(* Logix 5000 project; controller PRU vendor 1 type 14 code 107 rev 20.13; software revision 20.01 *)

TASK FeatureAdd1 (periodic, rate 10 ms, priority 10, watchdog 500 ms)
TASK INTERRUPT (periodic, rate 10 ms, priority 1, watchdog 200 ms) : SCREW_CONTROL
TASK MainTask (continuous, watchdog 500 ms) : MainProgram
TASK MSG (periodic, rate 500 ms, priority 10, watchdog 500 ms) : MSG
TASK Totalizers (periodic, rate 1000 ms, priority 3, watchdog 500 ms) : Totalizers

MODULES
   Local : vendor 1 type 14 code 107 (Compact 0, rev 20.13)
      LDI_2 : vendor 1 type 7 code 82 (Compact 15, rev 1.1, Input RPI 20 ms)
      LDI_1 : vendor 1 type 7 code 82 (Compact 14, rev 1.1, Input RPI 20 ms)
      ENCL : 1769-IQ16 (Compact 9, rev 1.1, Input RPI 2 ms)
      ENCR : 1769-IQ16 (Compact 10, rev 1.1, Input RPI 2 ms)
      LTC_3 : vendor 58 type 10 code 41 (Compact 8, rev 2.1, Input RPI 20 ms)
      LTC_4 : vendor 58 type 10 code 41 (Compact 11, rev 2.1, Input RPI 20 ms)
      LTC_2 : vendor 58 type 10 code 41 (Compact 7, rev 2.1, Input RPI 20 ms)
      LAO_1 : vendor 1 type 10 code 40 (Compact 4, rev 2.1, Output RPI 80 ms)
      LAI_1 : 1769-IF8 (Compact 1, rev 1.1, Output RPI 80 ms)
      LAI_2 : 1769-IF8 (Compact 2, rev 1.1, Output RPI 80 ms)
      LAO_2 : vendor 1 type 10 code 40 (Compact 5, rev 2.1, Output RPI 80 ms)
      LDO_2 : 1769-OB16 (Compact 13, rev 2.1, Output RPI 20 ms)
      LTC_1 : vendor 58 type 10 code 41 (Compact 6, rev 2.1, Input RPI 20 ms)
      LAI_3 : 1769-IF8 (Compact 3, rev 1.1, Output RPI 80 ms)
      LDO_1 : 1769-OB16 (Compact 12, rev 2.1, Output RPI 20 ms)
      IFS : vendor 1 type 14 code 107 (Ethernet 192.168.20.127, rev 20.1, $2b42fd4a$ RPI 500 ms)
      UTL_ENBT : 1768-ENBT (Ethernet 192.168.20.20, rev 4.1)
         UTL : vendor 1 type 14 code 74 (1768Ctrl5Slot 0, rev 20.1, $5e952958$ RPI 500 ms)
      CSS_A_ENBT : 1768-ENBT (Ethernet 192.168.20.70, rev 4.1)
         CSS_A : vendor 1 type 14 code 74 (1768Ctrl5Slot 0, rev 20.1, $71a6b3db$ RPI 500 ms)
      VFD_DRYERL : vendor 1 type 123 code 50 (Ethernet 192.168.20.112, rev 5.1, Output RPI 80 ms)
          : vendor 1 type 123 code 1535 (DPI 1, rev 6.1)
          : vendor 1 type 123 code 8192 (DPI 5, rev 4.2)
      VFD_DRYERR : vendor 1 type 123 code 50 (Ethernet 192.168.20.113, rev 5.1, Output RPI 80 ms)
          : vendor 1 type 123 code 1535 (DPI 1, rev 6.1)
          : vendor 1 type 123 code 8192 (DPI 5, rev 4.2)
      VFD_COOLSCREW : vendor 1 type 127 code 40 (Ethernet 192.168.20.114, rev 6.2, Output RPI 20 ms)
          : vendor 1 type 127 code 33792 (DSI 1, rev 1.8)
      IND560 : ETHERNET-MODULE (Ethernet 192.168.20.100, rev 1.1, Output RPI 100 ms)   // OutFeed Scale
END_MODULES

TYPE AnalogControl :
STRUCT
   AUTO : BOOL;   // 1=Auto, Control Requires automatic interlocks to enable the output
   MANUAL : BOOL;   // 1=Manual, Control (Forces the output Enable)
   MAN_SP : REAL;   // Sets the output in percent when the Manual bit is set
   AUTO_SP : REAL;   // Setpoint (usually provided by user) to control to when in Auto in Engineering Units
   CO : REAL;   // Control Output (%)
   FB : REAL;   // Feedback from the instrument (in Engineering units)
   PID_CO : REAL;   // Associated PID's Control Output (%)
   PV_SETPOINT : REAL;
   PV : REAL;   // Process Variable from measuring instrument (in Engineering units)
   HC_FAULT : BOOL;   // Controller Fault alarm bit
   RUN_STATUS : BOOL;   // Boolean feedback of the running status of the associated output
   START : BOOL;   // Master logical bit used to enable an associated output
   XA_Low : BOOL;   // Analog Signal failure (Low counts)
   XA_High : BOOL;   // Analog Signal failure (High counts)
   RawCounts : DINT;   // Raw integer from input card
   FailMode : DINT;   // In the event of a signal loss, 0=allow raw signal, 1=hold last good value, 2=hold at safe state value
   SafeState : REAL;   // Programatically set value to hold the signal to in case of a signal loss alarm
   AI_Anal : AI_Analysis;   // Used to manage an analog input to determine scaled value and loss of signal alarms
   InputMin : DINT;   // Input card lower counts i.e. 4mA - 4000 counts
   InputMax : DINT;   // Input card upper counts i.e. 20mA - 20000 counts
   ScaledMin : REAL;   // Analog low Engineering unit i.e. 4mA - 0 psi
   ScaledMax : REAL;   // Analog High Engineering unit i.e. 20mA - 100 psi
   OutputMin : DINT;   // Output card lower counts i.e. 4mA - 4000 counts
   OutputMax : DINT;   // Output card upper counts i.e. 4mA - 4000 counts
   AlarmsSetDetaults : BOOL;   // reloads the default alarm limits and setup
   Simulate : BOOL;   // 0=raw counts from Input card, 1=simulation raw counts
   RawCountsSim : DINT;   // raw count simulation from HMI/Programmer
   DifferenceExists : BOOL;   // 1 = A difference between default and current settings
   LoadDefaults : BOOL;   // set to 1=Load default values into the current values
   StoreDefaults : BOOL;   // set to 1=store the current setting values into the default settings
   AlarmDisable : BOOL;   // disables alarms 0=enabled 1=disabled
   PID_Enabled : BOOL;   // Tells the HMI if a PID exists
   mA : REAL;   // mA from Raw Counts
   AlarmWord : DINT;   // base2 alarm status
   Interlock : DINT;   // base2 Interlock Status
   HHEnabled : BOOL;
   HEnabled : BOOL;
   LEnabled : BOOL;
   LLEnabled : BOOL;
   Power : REAL;   // Current Power in kwatts
   Energy : REAL;   // Total Energy in kW-hr
   kWh_Tmr : TIMER;   // Energy Totalizer sample timer
   kWh_ResetPB : BOOL;   // HMI Reset Energy totals
   kWh_SampleTime : REAL;   // in seconds
   kWh_TimeMultiplier : REAL;   // derived from the SampleTime to ensure kW-Hr units
   PowerMax : REAL;   // Max Power Limit (kW)
END_STRUCT
END_TYPE

TYPE DateTime :   // Date and TimeOfDay (absolute) or Time (duration/interval)
STRUCT
   Yr : DINT;   // Year(s)
   Mo : DINT;   // Month(s)
   Da : DINT;   // Day(s)
   Hr : DINT;   // Hour(s)
   Min : DINT;   // Minute(s)
   Sec : DINT;   // Second(s)
   uSec : DINT;   // Microsecond(s)
END_STRUCT
END_TYPE

TYPE DUAL_SCREW :
STRUCT
   RPM_Setpoint : REAL;
   MODE_SCREW_AUTO : BOOL;
   MODE_SCREW_MAN : BOOL;
   MODE_SCREW_OFF : BOOL;
   MODE_SCREW : INT;
   SHUTDOWN_FAULTS_IOK : BOOL;
   HMI_AUTO_START_SCREW_PB : BOOL;
   HMI_STOP_SCREW_PB : BOOL;
   CMD_LEFT_SCREW_START : BOOL;
   CMD_LEFT_SCREW_STOP : BOOL;
   CMD_LEFT_SCREW_FWD : BOOL;
   CMD_LEFT_SCREW_REV : BOOL;
   CMD_RIGHT_SCREW_START : BOOL;
   CMD_RIGHT_SCREW_STOP : BOOL;
   CMD_RIGHT_SCREW_FWD : BOOL;
   CMD_RIGHT_SCREW_REV : BOOL;
   HMI_AUTO_SCREW_CMD_PCNT : REAL;
   AUTO_SCREW_LEFT_CMD_FREQ : REAL;
   AUTO_SCREW_MAX_PCNT : REAL;
   RPM_FREQ_MULTIPLIER : REAL;
   WIPER_OSC_INDEX : REAL;
   WIPER_OSC_SETPOINT : REAL;
   WIPER_OSC_AMPLITUDE : REAL;
   AUTO_SCREW_RIGHT_CMD_PCNT : REAL;
   AUTO_SCREW_RIGHT_CMD_FREQ : REAL;
   LEFT_ENCODER_G : INT;
   LEFT_ENCODER_BIN : DINT;
   RIGHT_ENCODER_G : INT;
   RIGHT_ENCODER_BIN : DINT;
   LEFT_ENCODER_TEMP : REAL;
   LEFT_ENCODER_DEG_IS : REAL;
   LEFT_ENCODER_DEG_WAS : REAL;
   RIGHT_ENCODER_TEMP : REAL;
   RIGHT_ENCODER_DEG_IS : REAL;
   RIGHT_ENCODER_DEG_WAS : REAL;
   LEFT_RIGHT_ENCODER_ERROR_TEMP : REAL;
   LEFT_RIGHT_ENCODER_ERROR_DEG : REAL;
   LEFT_ENCODER_DEG_WAS_SCANRATE : REAL;
   LEFT_ENCODER_DEG_WAS_SCANRATE_MOVED : REAL;
   RIGHT_ENCODER_DEG_WAS_SCANRATE : REAL;
   RIGHT_ENCODER_DEG_WAS_SCANRATE_MOVED : REAL;
   FINAL_SCREW_POSITION_ERROR : REAL;
   RIGHT_SCREW_RPM_COMPENSATION_GAIN : REAL;
   RIGHT_SCREW_RPM_COMP_PER_DEGREE : REAL;
   LEFT_AUTO_PCNT_SETPOINT : REAL;
   RIGHT_MAX_COMP_PCNT : REAL;
   RIGHT_MIN_COMP_PCNT : REAL;
END_STRUCT
END_TYPE

TYPE EnergyTot :   // Energy Totalizer
STRUCT
   EI : REAL;   // Current Amps
   Power : REAL;   // Current Power in kwatts
   Energy : REAL;   // Total Energy in kW-hr
   kWh_Tmr : TIMER;   // Energy Totalizer sample timer
   kWh_ResetPB : BOOL;   // HMI Reset Energy totals
   kWh_SampleTime : REAL;   // in seconds
   kWh_TimeMultiplier : REAL;   // derived from the SampleTime to ensure kW-Hr units
END_STRUCT
END_TYPE

TYPE FAULTRECORD :
STRUCT
   TIMELOW : DINT;
   TIMEHIGH : DINT;
   TYPE : INT;
   CODE : INT;
   INFO : DINT[8];
END_STRUCT
END_TYPE

TYPE KPI :   // Key Performance Indicators
STRUCT
   PowerTotal : REAL;   // Realtime total power consumption (kW)
   PowerPumps : REAL;   // Realtime pump power consumption (kW)
   PowerHeaters : REAL;   // Realtime heater power consumption (kW)
   PowerMisc : REAL;   // Realtime miscelaneous power consumption (kW)
   EnergyTotal : REAL;   // Energy Consumed Totalization (kW*hr)
   EnergyPumps : REAL;   // Energy Consumed pump total (kW*hr)
   EnergyHeaters : REAL;   // Energy Consumed heater total (kW*hr)
   EnergyMisc : REAL;   // Energy Consumed misc total (kW*hr)
   ProductVolTotal : REAL;   // Total product produced (US gal)
   ProductVolOil : REAL;   // Total heavy oil produced (US gal)
   ProductVolLightFraction : REAL;   // Total light fraction produced (US gal)
   WaterBleedTotal : REAL;   // Total water bled (US gal)
   WaterMakeupTotal : REAL;   // Total water made up (US gal)
   WaterFromFeedTotal : REAL;   // Total water from feed (US gal)
   FeedTotal : REAL;   // Total Feed (lbs)
   ProcessResidualTotal : REAL;   // Total Process Residual (lbs)
END_STRUCT
END_TYPE

TYPE MAJOR_FAULT :
STRUCT
   TYPE : INT;
   CODE : INT;
   INFO : DINT[8];
END_STRUCT
END_TYPE

TYPE PLCStatusData :   // Alarm and Status Data
STRUCT
   PLCSenonds : DINT;   // PLC Clock (Seconds) Used for Comms Loss
   AlarmMaster : DINT;   // Alarm Master
   SW_Status : DINT;   // Software Status
   HW_Statuts : DINT;   // Hardware Status
   CommsWarnSecSP : DINT;   // Comms Warning Time Setpoint
   CommsLossSecSP : DINT;   // Comms Loss Time Setpoint
   HousePowerOK : BOOL;   // House Power Ok
   GeneratorOk : BOOL;   // Generator Ok
   FireFlowAlm : BOOL;   // FIRE SYSTEM FLOW Alarm
   OptionH3 : BOOL;   // OPTION H3 OCCUPANCY 0=DISABLED 1=ENABLED
   Status : DINT[10];   // Status Data
END_STRUCT
END_TYPE

TYPE SystemAlarmMonitor :
STRUCT
   AlarmMaster : DINT;   // b0=msg b1=warn b2=CSS_Start_Disable b3=PRU_Strt_Disable b4=PRU_Run_Disable
   AlarmDisablePB : BOOL;   // set to 1 to toggle the AlarmDisable bit
   AlarmDisablePB_Toggle : PB_Toggle;
   AlarmDisabled : BOOL;   // 1=ignore system alarms
   AlarmDisableTmr : TIMER;
   AlarmDisableTimeOut : DINT;   // in minutes
   AlarmDisableMaxTimeAlm : BOOL;   // Max time has elabsed. Alert User of alarm condition
   Alm_Message : BOOL;   // Message Alarm Exists
   Alm_Warning : BOOL;   // Warning Alarm Exist
   Alm_CSS_Start_Disable : BOOL;   // CSS_Start_Disable Alarm Exists
   Alm_PRU_Start_Disable : BOOL;   // PRU_Start_Disable Alarm Exists
   Alm_PRU_Run_Disable : BOOL;   // PRU_Run_Disable Alarm Exists
   CommsErrorTmr : TIMER;
   CommsLossTmr : TIMER;
   LossOfComms : BOOL;   // 1=alarm
   CommsError : BOOL;   // 1=alarm
   CommsStatus : DINT;   // 0=Ok 1=CommsError 2=Loss of Comms
   CommsMaster : DINT[4];   // General Status
   AlmTmr : TIMER[5];
   Heartbeat : DINT;   // seconds
   HeartbeatLast : DINT;   // seconds
   ReadWord : DINT[11];   // [0]=Heartbeat [1]=AlarmMaster [2]=status...
END_STRUCT
END_TYPE

TYPE VFD :   // Variable Frequency Data Type.
STRUCT
   HMI_MODE_OFF_PB : BOOL;
   HMI_MODE_MAINT_PB : BOOL;
   HMI_MODE_SEMI_PB : BOOL;
   HMI_MODE_AUTO_PB : BOOL;
   MODE : INT;
   HMI_FWD_PB : BOOL;
   HMI_REV_PB : BOOL;
   HMI_JOG_FWD_PB : BOOL;
   HMI_JOG_REV_PB : BOOL;
   HMI_START_AUTO_PB : BOOL;
   HMI_STOP_PB : BOOL;
   SPEED_SETPOINT_SEMI : REAL;
   SPEED_SETPOINT_AUTO : REAL;
   INTERLOCK_1 : BOOL;
   INTERLOCK_2 : BOOL;
   INTERLOCK_3 : BOOL;
   ACTUAL_ENABLED : BOOL;
   ACTUAL_SPEED : REAL;
   ACTUAL_SPEED_CONVERSION_FACTOR : REAL;
   MODE_OFF_ION : BOOL;
   MODE_MAINT_ION : BOOL;
   MODE_SEMI_ION : BOOL;
   MODE_AUTO_ION : BOOL;
   VFD_BEEN_ON : BOOL;
   VFD_BEEN_OFF : BOOL;
   CMD_STOPPED : BOOL;
   CMD_AUTO_RUN_ENABLED : BOOL;
   CMD_AUTO_STARTED : BOOL;
END_STRUCT
END_TYPE

ADD_ON_INSTRUCTION AI_1769_IF4   (* revision 1.0, vendor Deterministic Systems, Inc. *)
// Analog Input Conversion
VAR_INPUT
   IN_ANALOG_INPUT_RAW : INT; {required}
   IN_Ai_Lo_Scale : REAL; {required}
   IN_Ai_Hi_Scale : REAL; {required}
   IN_HMI_AI_FORCE : BOOL; {required}
   IN_HMI_Ai_FORCE_VALUE : REAL; {required}
END_VAR
VAR_OUTPUT
   OUT_Ai_Calc : REAL; {access Read Only, required}
   OUT_ANALOG_OUTPUT : REAL; {access Read Only, required}
END_VAR
VAR
   Ai_Raw : REAL; {access None}
   Ai_M : REAL; {access None}
   Ai_B : REAL; {access None}
   Ai_INPUT : REAL; {access None}
END_VAR

ROUTINE Logic   (* ladder *)
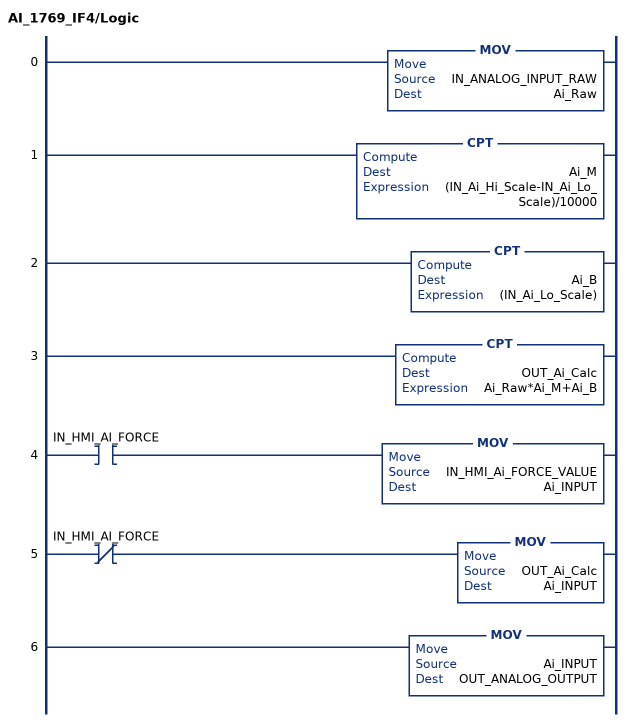
   0: MOV(IN_ANALOG_INPUT_RAW,Ai_Raw);
   1: CPT(Ai_M,(IN_Ai_Hi_Scale-IN_Ai_Lo_Scale)/10000);
   2: CPT(Ai_B,(IN_Ai_Lo_Scale));
   3: CPT(OUT_Ai_Calc,Ai_Raw*Ai_M+Ai_B);
   4: XIC(IN_HMI_AI_FORCE)MOV(IN_HMI_Ai_FORCE_VALUE,Ai_INPUT);
   5: XIO(IN_HMI_AI_FORCE)MOV(OUT_Ai_Calc,Ai_INPUT);
   6: MOV(Ai_INPUT,OUT_ANALOG_OUTPUT);
END_ROUTINE
END_ADD_ON_INSTRUCTION

ADD_ON_INSTRUCTION AI_Analysis   (* revision 1.0 *)
VAR_OUTPUT
   XmtrOut : REAL; {access Read Only, required}
END_VAR
VAR_INPUT
   RawCounts : DINT; {required}
   SafeState : REAL; {required}
END_VAR
VAR_OUTPUT
   SigLossHigh : BOOL; {required}
   SigLossLow : BOOL; {required}
END_VAR
VAR_INPUT
   FailMode : DINT; {required}   // 0=raw, 1=last state, 2=safe state
   SigLossHighSP : DINT; {required}
   SigLossLowSP : DINT; {required}
   InputMin : REAL; {required}
   InputMax : REAL; {required}
   ScaledMin : REAL; {required}
   ScaledMax : REAL; {required}
   Simulate : BOOL; {required}
   RawCountsSim : DINT; {access None, required}
END_VAR
VAR_OUTPUT
   mA : REAL; {access Read Only, required}
END_VAR
VAR
   SigLoss : BOOL; {access None}
   LastState : REAL; {access None}
   MyXmtrSCP : SCLP; {access None}
   MyRawCounts : DINT; {access None}
END_VAR

ROUTINE Logic   (* ladder *)
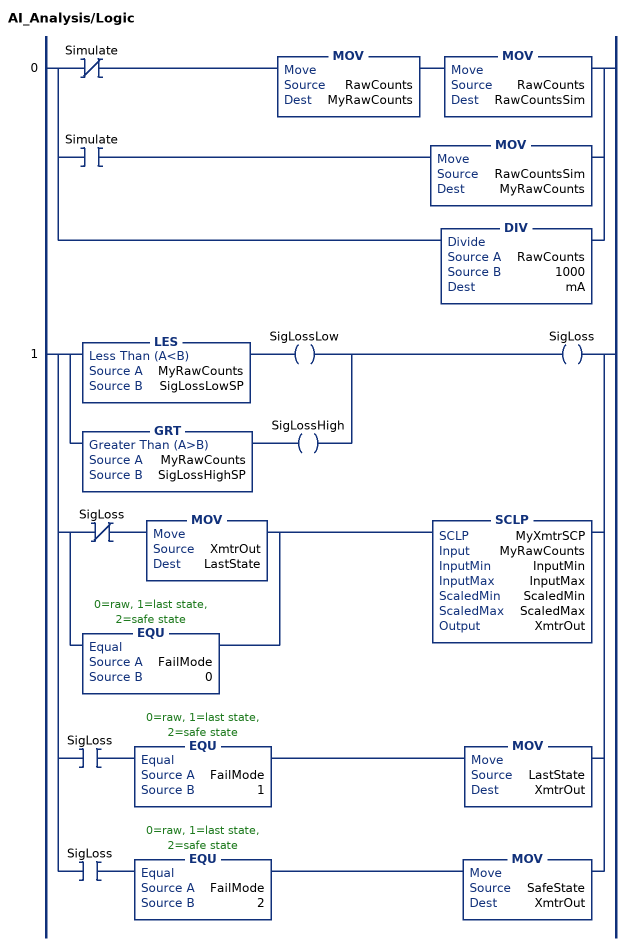
   0: [XIO(Simulate) MOV(RawCounts,MyRawCounts) MOV(RawCounts,RawCountsSim) ,XIC(Simulate) MOV(RawCountsSim,MyRawCounts) ,DIV(RawCounts,1000,mA) ];
   1: [[LES(MyRawCounts,SigLossLowSP) OTE(SigLossLow) ,GRT(MyRawCounts,SigLossHighSP) OTE(SigLossHigh) ] OTE(SigLoss) ,[XIO(SigLoss) MOV(XmtrOut,LastState) ,EQU(FailMode,0) ] SCLP(MyXmtrSCP,MyRawCounts,InputMin,InputMax,ScaledMin,ScaledMax,XmtrOut) ,XIC(SigLoss) EQU(FailMode,1) MOV(LastState,XmtrOut) ,XIC(SigLoss) EQU(FailMode,2) MOV(SafeState,XmtrOut) ];
END_ROUTINE
END_ADD_ON_INSTRUCTION

ADD_ON_INSTRUCTION AI_Totalizer   (* revision 1.0 *)
// Flow Totalizer
VAR_INPUT
   Input : REAL; {access Read Only, required}   // Input to Totalize
   Midnight : BOOL; {access Read Only, required}   // Midnight Input Trigger
   SampleTimerSP : DINT; {required}   // Sample Interval
   TimeBase : DINT; {required}   // Type 1 = Per Second 2 = Per Minute 3 = Per Hour 4 = Per Day
   MinimumInc : REAL; {required}   // Mimimum Totalizer Increment
   IDP : DINT; {required}   // Implied Decimal Point
   RollOver : DINT := 9999999; {access Read Only, required}   // Roll Over Value
END_VAR
VAR_OUTPUT
   NonResetTotal : DINT; {access Read Only, visible}   // Non Resetable Totalized Value
   TodayTotal : DINT; {access Read Only, visible}   // Todays Total
   YestTotal : DINT; {access Read Only, visible}   // Yesterdays Total
   ResetTotal : DINT; {access Read Only, visible}   // Resetable Totalized Value
END_VAR
VAR_INPUT
   Reset : BOOL;   // Reset Input
END_VAR
VAR
   UpdateTotValues : BOOL; {access None}   // Update Totalized Values
   Timer : DINT; {access None}   // Timer Value
   TestONS : BOOL; {access None}
   SamplePulse : BOOL; {access None}   // Sample Pulse
   OneShot : BOOL; {access None}
   ModRemain : REAL; {access None}
   InputPerSampleWhole : DINT; {access None}
   InputPerSampleBuff : REAL; {access None}   // Input Value Per Sample High Accuracy Buffer
   InputPerSample : REAL; {access None}
   InputInSecond : REAL; {access None}
   InputIDPOffSet : REAL; {access None}
   IDPOffSet : DINT; {access None}   // IDP Offset
END_VAR

ROUTINE Logic   (* ladder *)
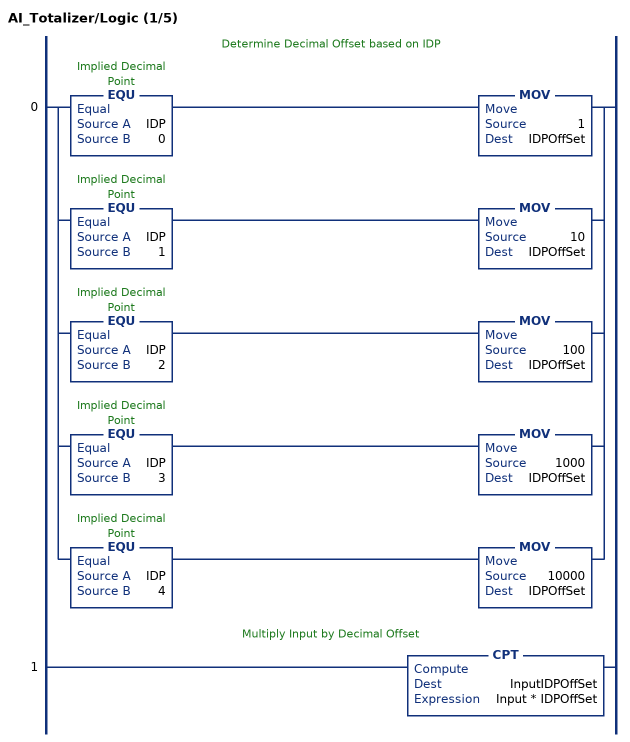
   // Determine Decimal Offset based on IDP
   0: [EQU(IDP,0) MOV(1,IDPOffSet) ,EQU(IDP,1) MOV(10,IDPOffSet) ,EQU(IDP,2) MOV(100,IDPOffSet) ,EQU(IDP,3) MOV(1000,IDPOffSet) ,EQU(IDP,4) MOV(10000,IDPOffSet) ];
   // Multiply Input by Decimal Offset
   1: CPT(InputIDPOffSet,Input * IDPOffSet);
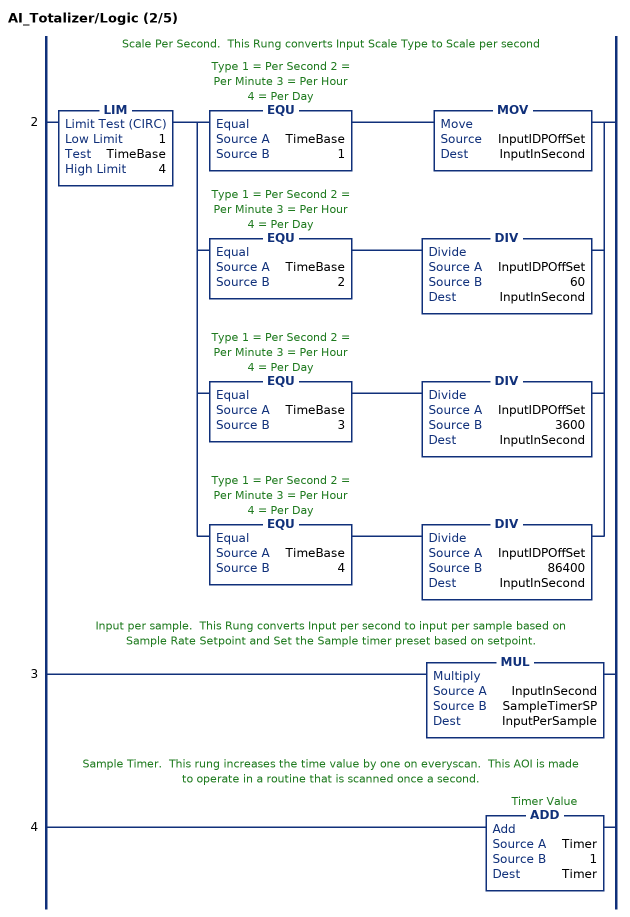
   // Scale Per Second.  This Rung converts Input Scale Type to Scale per second
   2: LIM(1,TimeBase,4)[EQU(TimeBase,1) MOV(InputIDPOffSet,InputInSecond) ,EQU(TimeBase,2) DIV(InputIDPOffSet,60,InputInSecond) ,EQU(TimeBase,3) DIV(InputIDPOffSet,3600,InputInSecond) ,EQU(TimeBase,4) DIV(InputIDPOffSet,86400,InputInSecond) ];
   // Input per sample.  This Rung converts Input per second to input per sample based on Sample Rate Setpoint and Set the Sample timer preset based on setpoint.
   3: MUL(InputInSecond,SampleTimerSP,InputPerSample);
   // Sample Timer.  This rung increases the time value by one on everyscan.  This AOI is made to operate in a routine that is scanned once a second.
   4: ADD(Timer,1,Timer);
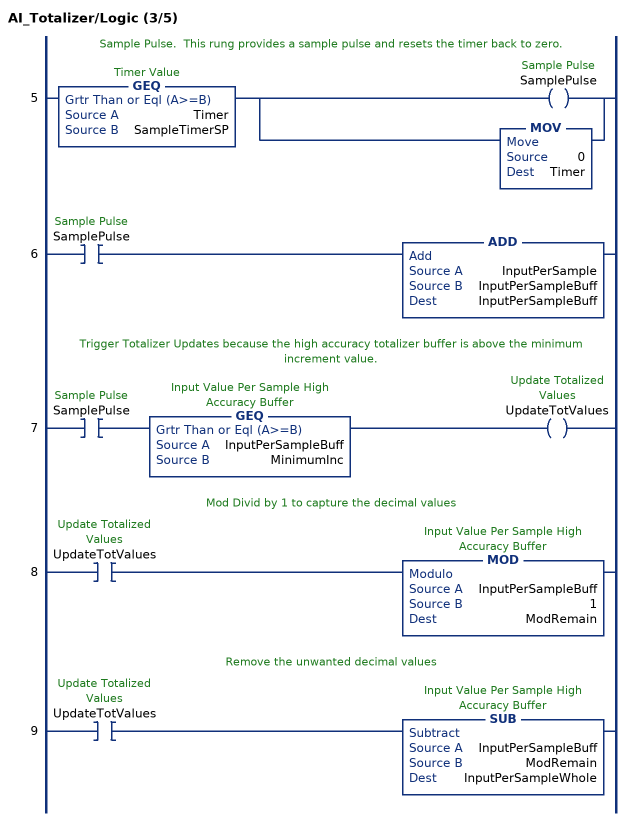
   // Sample Pulse.  This rung provides a sample pulse and resets the timer back to zero.
   5: GEQ(Timer,SampleTimerSP)[OTE(SamplePulse) ,MOV(0,Timer) ];
   6: XIC(SamplePulse)ADD(InputPerSample,InputPerSampleBuff,InputPerSampleBuff);
   // Trigger Totalizer Updates because the high accuracy totalizer buffer is above the minimum increment value.
   7: XIC(SamplePulse)GEQ(InputPerSampleBuff,MinimumInc)OTE(UpdateTotValues);
   // Mod Divid by 1 to capture the decimal values
   8: XIC(UpdateTotValues)MOD(InputPerSampleBuff,1,ModRemain);
   // Remove the unwanted decimal values
   9: XIC(UpdateTotValues)SUB(InputPerSampleBuff,ModRemain,InputPerSampleWhole);
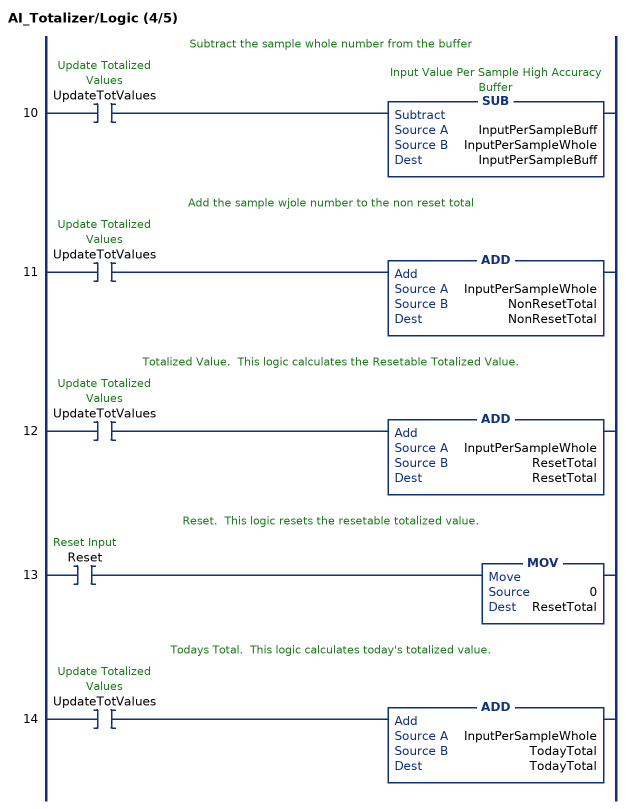
   // Subtract the sample whole number from the buffer
   10: XIC(UpdateTotValues)SUB(InputPerSampleBuff,InputPerSampleWhole,InputPerSampleBuff);
   // Add the sample wjole number to the non reset total
   11: XIC(UpdateTotValues)ADD(InputPerSampleWhole,NonResetTotal,NonResetTotal);
   // Totalized Value.  This logic calculates the Resetable Totalized Value.
   12: XIC(UpdateTotValues)ADD(InputPerSampleWhole,ResetTotal,ResetTotal);
   // Reset.  This logic resets the resetable totalized value.
   13: XIC(Reset)MOV(0,ResetTotal);
   // Todays Total.  This logic calculates today's totalized value.
   14: XIC(UpdateTotValues)ADD(InputPerSampleWhole,TodayTotal,TodayTotal);
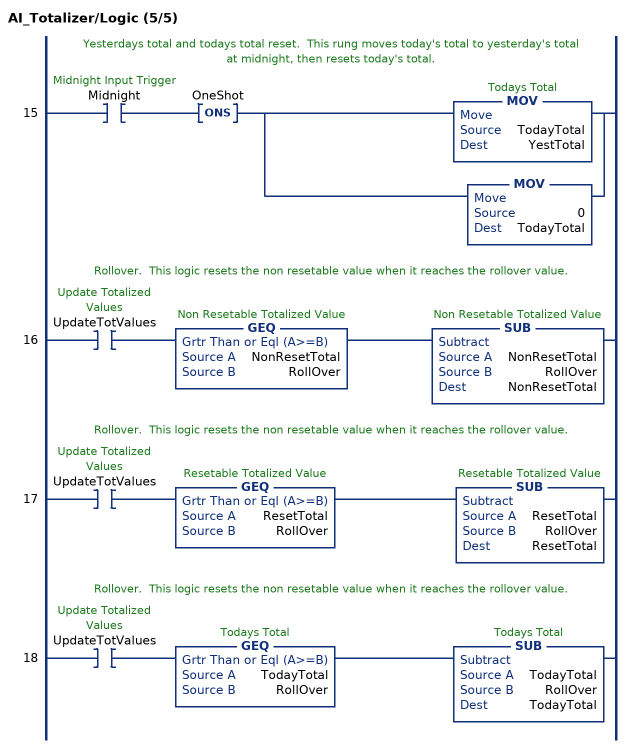
   // Yesterdays total and todays total reset.  This rung moves today's total to yesterday's total at midnight, then resets today's total.
   15: XIC(Midnight)ONS(OneShot)[MOV(TodayTotal,YestTotal) ,MOV(0,TodayTotal) ];
   // Rollover.  This logic resets the non resetable value when it reaches the rollover value.
   16: XIC(UpdateTotValues)GEQ(NonResetTotal,RollOver)SUB(NonResetTotal,RollOver,NonResetTotal);
   // Rollover.  This logic resets the non resetable value when it reaches the rollover value.
   17: XIC(UpdateTotValues)GEQ(ResetTotal,RollOver)SUB(ResetTotal,RollOver,ResetTotal);
   // Rollover.  This logic resets the non resetable value when it reaches the rollover value.
   18: XIC(UpdateTotValues)GEQ(TodayTotal,RollOver)SUB(TodayTotal,RollOver,TodayTotal);
END_ROUTINE
END_ADD_ON_INSTRUCTION

ADD_ON_INSTRUCTION DSi_5050_PULSE   (* revision 1.0, vendor Deterministic Systems, Inc. *)
// Pulse Ouput with 50% duty cycle.
VAR_INPUT
   MS : DINT := 1000; {access None, required}
   IN_ENABLE : BOOL; {required}
END_VAR
VAR_OUTPUT
   OUT_5050_SS : BOOL; {access Read Only, required}
   OUT_5050 : BOOL; {access Read Only, required}
END_VAR
VAR
   ONE_SEC_TONA : TIMER := (PRE := 500, ACC := 485); {access None}
   ONE_SEC_TONB : TIMER := (PRE := 500); {access None}
   OUT_5050_ONS : BOOL; {access None}
END_VAR

ROUTINE Logic   (* ladder *)
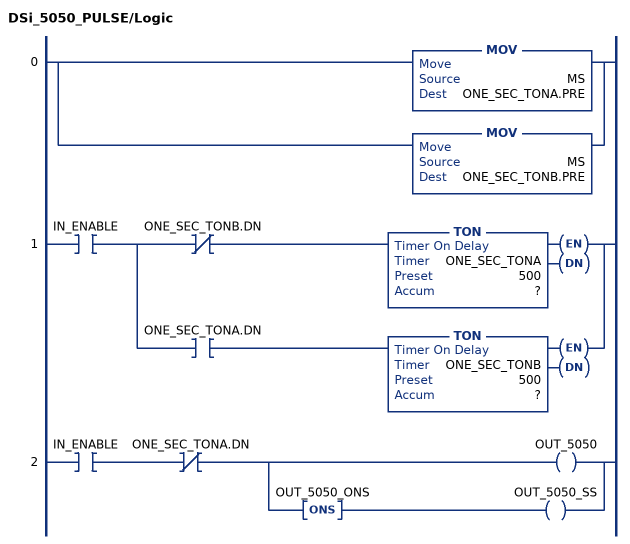
   0: [MOV(MS,ONE_SEC_TONA.PRE) ,MOV(MS,ONE_SEC_TONB.PRE) ];
   1: XIC(IN_ENABLE)[XIO(ONE_SEC_TONB.DN) TON(ONE_SEC_TONA,?,?) ,XIC(ONE_SEC_TONA.DN) TON(ONE_SEC_TONB,?,?) ];
   2: XIC(IN_ENABLE)XIO(ONE_SEC_TONA.DN)[OTE(OUT_5050) ,ONS(OUT_5050_ONS) OTE(OUT_5050_SS) ];
END_ROUTINE
END_ADD_ON_INSTRUCTION

ADD_ON_INSTRUCTION DSi_COMP_SCALE   (* revision 1.1, vendor Deterministic Systems, Inc. *)
// Rate of Change
VAR_INPUT
   IN_VALUE_END : REAL; {required}
   IN_INC_VALUE : REAL; {required}
END_VAR
VAR_OUTPUT
   OUT_VALUE : REAL; {access Read Only, required}
   OUT_COMP : REAL; {access Read Only, required}
END_VAR
VAR
   TEMP_VALUE : REAL; {access None}
   VALUE_WAS_GRT : BOOL; {access None}
   TEMP_COMP : REAL; {access None}
END_VAR

ROUTINE Logic   (* ladder *)
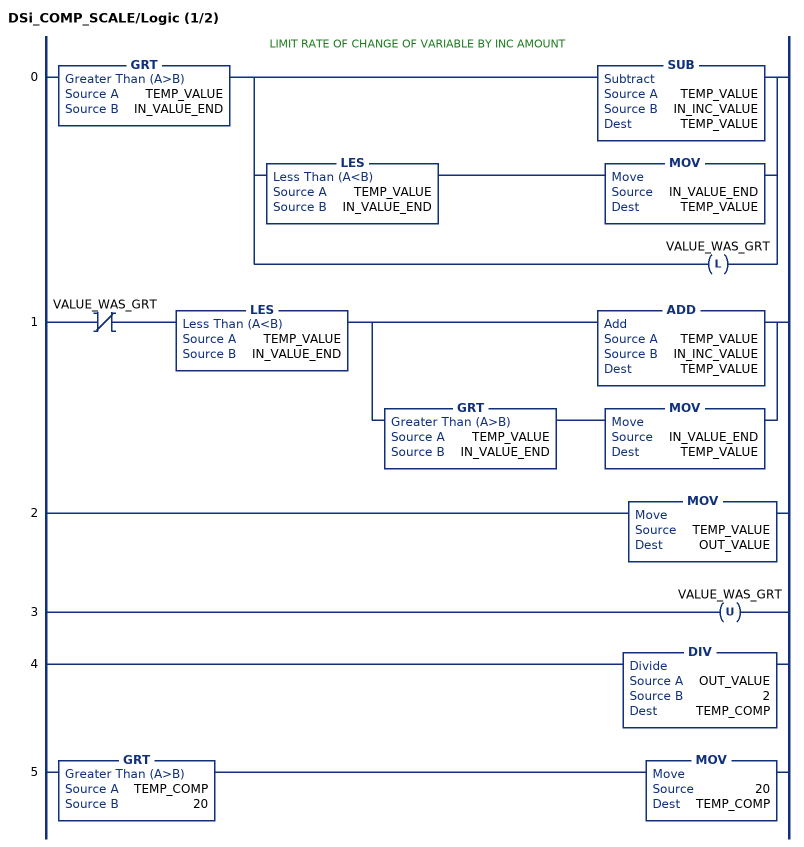
   // LIMIT RATE OF CHANGE OF VARIABLE BY INC AMOUNT
   0: GRT(TEMP_VALUE,IN_VALUE_END)[SUB(TEMP_VALUE,IN_INC_VALUE,TEMP_VALUE) ,LES(TEMP_VALUE,IN_VALUE_END) MOV(IN_VALUE_END,TEMP_VALUE) ,OTL(VALUE_WAS_GRT) ];
   1: XIO(VALUE_WAS_GRT)LES(TEMP_VALUE,IN_VALUE_END)[ADD(TEMP_VALUE,IN_INC_VALUE,TEMP_VALUE) ,GRT(TEMP_VALUE,IN_VALUE_END) MOV(IN_VALUE_END,TEMP_VALUE) ];
   2: MOV(TEMP_VALUE,OUT_VALUE);
   3: OTU(VALUE_WAS_GRT);
   4: DIV(OUT_VALUE,2,TEMP_COMP);
   5: GRT(TEMP_COMP,20)MOV(20,TEMP_COMP);
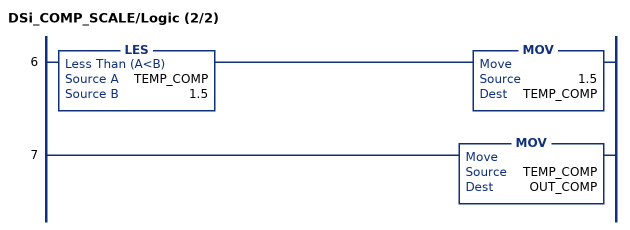
   6: LES(TEMP_COMP,1.5)MOV(1.5,TEMP_COMP);
   7: MOV(TEMP_COMP,OUT_COMP);
END_ROUTINE
END_ADD_ON_INSTRUCTION

ADD_ON_INSTRUCTION DSi_WF50   (* revision 1.0, vendor Deterministic Systems, Inc. *)
// Walking Filter - 10 elements.
VAR_INPUT
   IN_VALUE : REAL; {required}
END_VAR
VAR_OUTPUT
   OUT_VALUE : REAL; {access Read Only, required}
END_VAR
VAR
   INDEX : INT; {access None}
   DATA_TOTAL : REAL; {access None}
   DATA : REAL[51]; {access None}
END_VAR

ROUTINE Logic   (* ladder *)
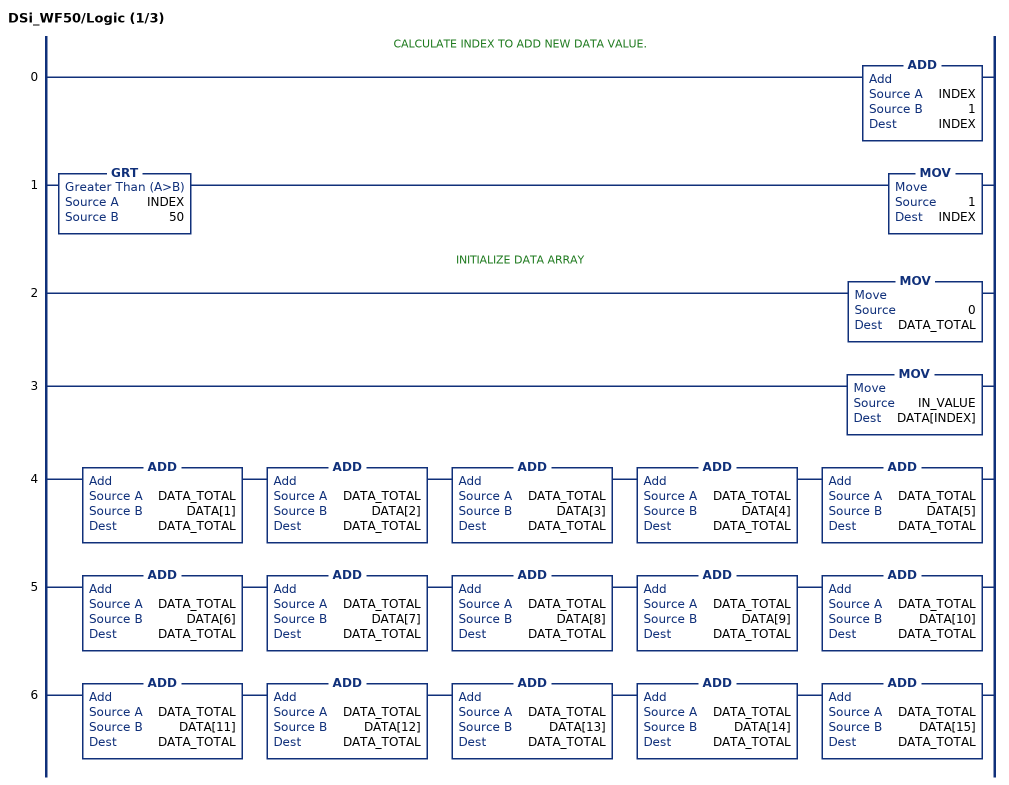
   // CALCULATE INDEX TO ADD NEW DATA VALUE.
   0: ADD(INDEX,1,INDEX);
   1: GRT(INDEX,50)MOV(1,INDEX);
   // INITIALIZE DATA ARRAY
   2: MOV(0,DATA_TOTAL);
   3: MOV(IN_VALUE,DATA[INDEX]);
   4: ADD(DATA_TOTAL,DATA[1],DATA_TOTAL)ADD(DATA_TOTAL,DATA[2],DATA_TOTAL)ADD(DATA_TOTAL,DATA[3],DATA_TOTAL)ADD(DATA_TOTAL,DATA[4],DATA_TOTAL)ADD(DATA_TOTAL,DATA[5],DATA_TOTAL);
   5: ADD(DATA_TOTAL,DATA[6],DATA_TOTAL)ADD(DATA_TOTAL,DATA[7],DATA_TOTAL)ADD(DATA_TOTAL,DATA[8],DATA_TOTAL)ADD(DATA_TOTAL,DATA[9],DATA_TOTAL)ADD(DATA_TOTAL,DATA[10],DATA_TOTAL);
   6: ADD(DATA_TOTAL,DATA[11],DATA_TOTAL)ADD(DATA_TOTAL,DATA[12],DATA_TOTAL)ADD(DATA_TOTAL,DATA[13],DATA_TOTAL)ADD(DATA_TOTAL,DATA[14],DATA_TOTAL)ADD(DATA_TOTAL,DATA[15],DATA_TOTAL);
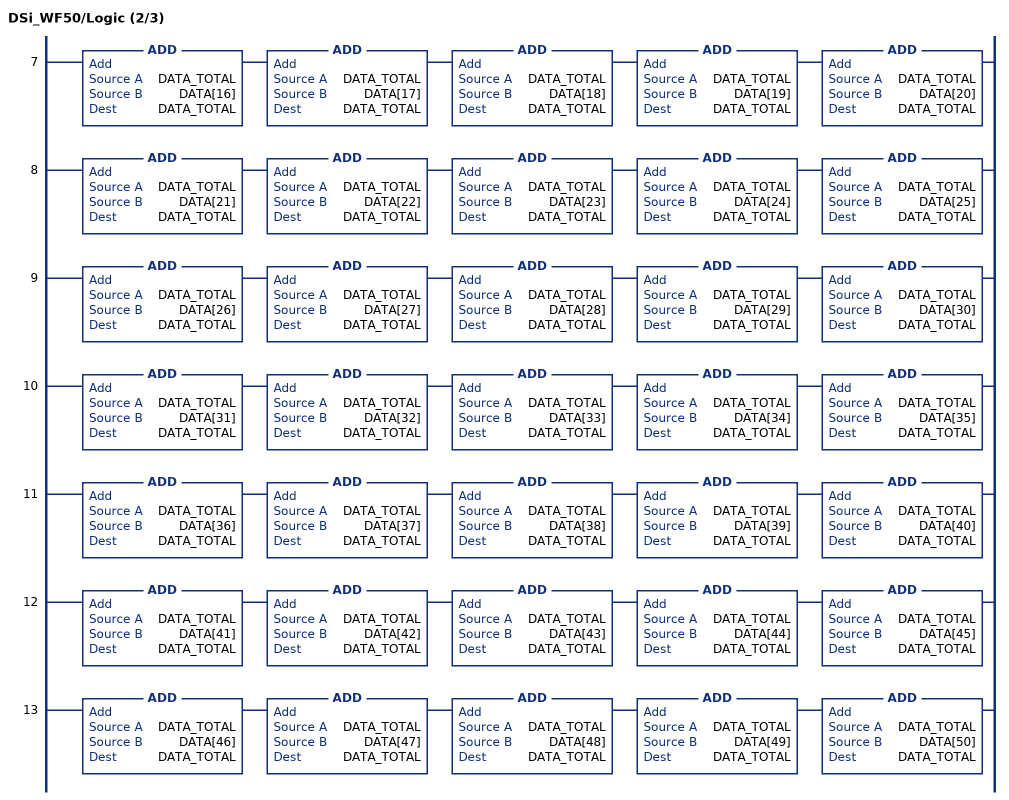
   7: ADD(DATA_TOTAL,DATA[16],DATA_TOTAL)ADD(DATA_TOTAL,DATA[17],DATA_TOTAL)ADD(DATA_TOTAL,DATA[18],DATA_TOTAL)ADD(DATA_TOTAL,DATA[19],DATA_TOTAL)ADD(DATA_TOTAL,DATA[20],DATA_TOTAL);
   8: ADD(DATA_TOTAL,DATA[21],DATA_TOTAL)ADD(DATA_TOTAL,DATA[22],DATA_TOTAL)ADD(DATA_TOTAL,DATA[23],DATA_TOTAL)ADD(DATA_TOTAL,DATA[24],DATA_TOTAL)ADD(DATA_TOTAL,DATA[25],DATA_TOTAL);
   9: ADD(DATA_TOTAL,DATA[26],DATA_TOTAL)ADD(DATA_TOTAL,DATA[27],DATA_TOTAL)ADD(DATA_TOTAL,DATA[28],DATA_TOTAL)ADD(DATA_TOTAL,DATA[29],DATA_TOTAL)ADD(DATA_TOTAL,DATA[30],DATA_TOTAL);
   10: ADD(DATA_TOTAL,DATA[31],DATA_TOTAL)ADD(DATA_TOTAL,DATA[32],DATA_TOTAL)ADD(DATA_TOTAL,DATA[33],DATA_TOTAL)ADD(DATA_TOTAL,DATA[34],DATA_TOTAL)ADD(DATA_TOTAL,DATA[35],DATA_TOTAL);
   11: ADD(DATA_TOTAL,DATA[36],DATA_TOTAL)ADD(DATA_TOTAL,DATA[37],DATA_TOTAL)ADD(DATA_TOTAL,DATA[38],DATA_TOTAL)ADD(DATA_TOTAL,DATA[39],DATA_TOTAL)ADD(DATA_TOTAL,DATA[40],DATA_TOTAL);
   12: ADD(DATA_TOTAL,DATA[41],DATA_TOTAL)ADD(DATA_TOTAL,DATA[42],DATA_TOTAL)ADD(DATA_TOTAL,DATA[43],DATA_TOTAL)ADD(DATA_TOTAL,DATA[44],DATA_TOTAL)ADD(DATA_TOTAL,DATA[45],DATA_TOTAL);
   13: ADD(DATA_TOTAL,DATA[46],DATA_TOTAL)ADD(DATA_TOTAL,DATA[47],DATA_TOTAL)ADD(DATA_TOTAL,DATA[48],DATA_TOTAL)ADD(DATA_TOTAL,DATA[49],DATA_TOTAL)ADD(DATA_TOTAL,DATA[50],DATA_TOTAL);
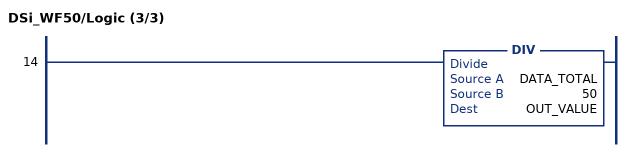
   14: DIV(DATA_TOTAL,50,OUT_VALUE);
END_ROUTINE
END_ADD_ON_INSTRUCTION

ADD_ON_INSTRUCTION MovingAve   (* revision 1.0 *)
VAR_INPUT
   InputData : REAL; {required}
   SampleRateTmrPRE : DINT; {required}
   Initialize : BOOL; {required}
   NumberOfSamples : DINT; {required}
END_VAR
VAR_IN_OUT
   OutputData : REAL; {required}
END_VAR
VAR
   MAVE_01 : MOVING_AVERAGE := (SampleEnable := 1, NumberOfSamples := 1);
   TONR_01 : FBD_TIMER;
   Storage : REAL[1000];
   MUL_01 : FBD_MATH;
   __l01CE2E511B44B3CD : BOOL;
   __l01CE5AF01B44D61A : REAL;
   __l01CE66631B44C5FE : DINT;
   __l01CE1ADE1B44D747 : DINT;
END_VAR

ROUTINE Logic   (* function block diagram *)
   SHEET 1
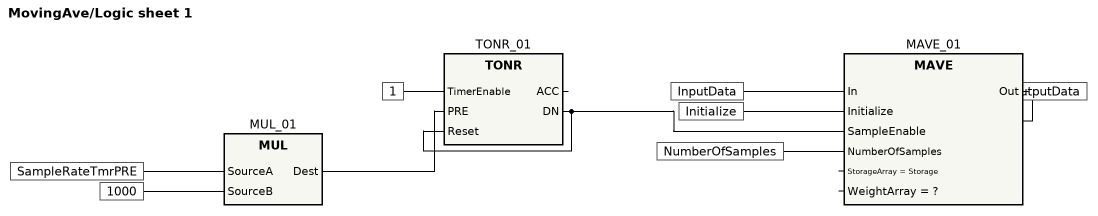
   MUL_01 : MUL(SourceA := SampleRateTmrPRE, SourceB := 1000);
   TONR_01 : TONR(TimerEnable := 1, PRE := MUL_01.Dest, Reset := TONR_01.DN);   // unwired pins: ACC
   MAVE_01 : MAVE(In := InputData, Initialize := Initialize, SampleEnable := TONR_01.DN, NumberOfSamples := NumberOfSamples, StorageArray := Storage, WeightArray := ?);
   OutputData := MAVE_01.Out;
END_ROUTINE
END_ADD_ON_INSTRUCTION

ADD_ON_INSTRUCTION PB_Toggle   (* revision 1.0, ExecuteEnableInFalse *)
// This AOI toggles a boolean tag (ie. DistPump1.Online) and resets the HMI PB.  Condition this rung with the HMI PB.
VAR_IN_OUT
   PB : BOOL; {required}
   Toggle : BOOL; {required}
END_VAR
VAR
   PBONS1 : BOOL;
   PB_Latch : BOOL;
END_VAR

ROUTINE EnableInFalse   (* ladder *)
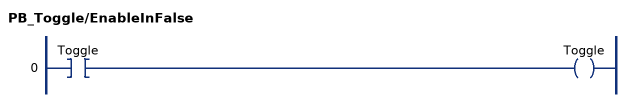
   0: XIC(Toggle)OTE(Toggle);
END_ROUTINE

ROUTINE Logic   (* ladder *)
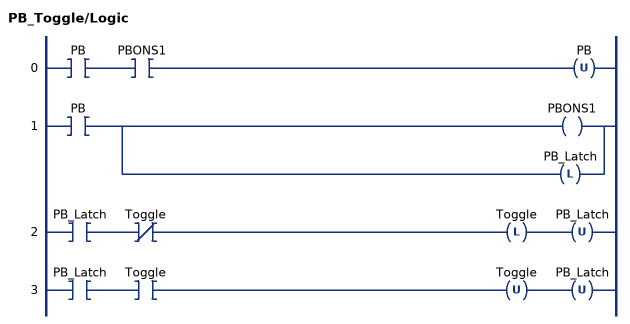
   0: XIC(PB)XIC(PBONS1)OTU(PB);
   1: XIC(PB)[OTE(PBONS1) ,OTL(PB_Latch) ];
   2: XIC(PB_Latch)XIO(Toggle)OTL(Toggle)OTU(PB_Latch);
   3: XIC(PB_Latch)XIC(Toggle)OTU(Toggle)OTU(PB_Latch);
END_ROUTINE
END_ADD_ON_INSTRUCTION

ADD_ON_INSTRUCTION SCLP   (* revision 1.0, vendor Rockwell Automation *)
VAR_INPUT
   Input : REAL; {required}
   InputMin : REAL; {required}
   InputMax : REAL; {required}
   ScaledMin : REAL; {required}
   ScaledMax : REAL; {required}
END_VAR
VAR_OUTPUT
   Output : REAL; {access Read Only, required}
END_VAR
VAR
   Temp1 : REAL;
   Temp2 : REAL;
   Rate : REAL;
   Temp4 : REAL;
   Offset : REAL;
   Temp3 : REAL;
END_VAR

ROUTINE Logic   (* ladder *)
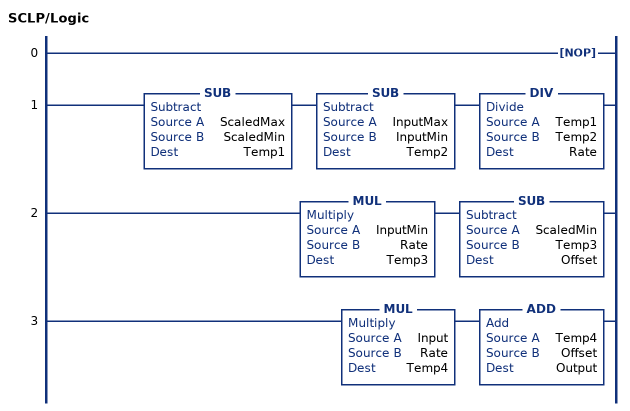
   0: NOP();
   1: SUB(ScaledMax,ScaledMin,Temp1)SUB(InputMax,InputMin,Temp2)DIV(Temp1,Temp2,Rate);
   2: MUL(InputMin,Rate,Temp3)SUB(ScaledMin,Temp3,Offset);
   3: MUL(Input,Rate,Temp4)ADD(Temp4,Offset,Output);
END_ROUTINE
END_ADD_ON_INSTRUCTION

ADD_ON_INSTRUCTION SCREW_ENCODERS   (* revision 1.1, vendor Deterministic Systems, Inc. *)
VAR_INPUT
   GS_LEFT_ENCODER_INT_IN : INT; {required}
   GS_RIGHT_ENCODER_INT_IN : INT; {required}
END_VAR
VAR_OUTPUT
   LEFT_ENCODER_DEG_OUT_REAL_OUT : REAL; {access Read Only, required}
   RIGHT_ENCODER_DEG_OUT_REAL_OUT : REAL; {access Read Only, required}
   LEFT_RIGHT_ENCODER_ERROR_DEG_REAL_OUT : REAL; {access Read Only, required}
   LEFT_ENCODER_DEG_WAS_SCANRATE_MOVED_OUT : REAL; {access Read Only, required}
   RIGHT_ENCODER_DEG_WAS_SCANRATE_MOVED_OUT : REAL; {access Read Only, required}
END_VAR
VAR_INPUT
   MASTER_RIGHT_BOOL_IN : BOOL; {required}
END_VAR
VAR_OUTPUT
   ENCODER_MOVED_LAST_SEC_REAL_OUT : REAL; {access Read Only, required}
   MIX_REV_PER_MIN_REAL_OUT : REAL; {access Read Only, required}
   RETENTION_TIME_MIN_REAL_OUT : REAL; {access Read Only, required}
END_VAR
VAR_INPUT
   MIX_FWD_PRESET_REAL_IN : REAL; {required}
   MIX_REV_PRESET_REAL_IN : REAL; {required}
END_VAR
VAR_OUTPUT
   AUTO_FWD_CMD_BOOL_OUT : BOOL; {access Read Only, required}
   ENCODER_ACC_REAL_OUT : REAL; {access Read Only, required}
END_VAR
VAR_INPUT
   SREW_MODE_INT_IN : INT; {required}
   SCREW_PITCH_CONSTANT_REAL_IN : REAL; {required}
   ENCODER_OFFSET_IN : REAL; {required}
END_VAR
VAR
   LEFT_ENCODER_BIN : DINT;
   LEFT_ENCODER_G : DINT;
   RIGHT_ENCODER_BIN : DINT;
   RIGHT_ENCODER_G : DINT;
   LEFT_ENCODER_TEMP : REAL;
   RIGHT_ENCODER_TEMP : REAL;
   LEFT_RIGHT_ENCODER_ERROR_TEMP : REAL;
   ENC_SCAN_COUNT : INT;
   MIX_SEQ : INT;
   ONE_SECOND_ENCODER_SCAN : BOOL;   // 100 x 10mS.
   LEFT_ENCODER_DEG_WAS_SCANRATE : REAL;
   RIGHT_ENCODER_DEG_WAS_SCANRATE : REAL;
   MIX_SEQ_STEP_00_DONE_TON : TIMER := (PRE := 100);
   MIX_SEQ_STEP_01_DONE : BOOL;
   MIX_SEQ_STEP_02_DONE : BOOL;
   MIX_STEP_00_ION : BOOL;
   MIX_STEP_01_ION : BOOL;   // FORWARD
   MIX_STEP_01_ONSN : BOOL;
   MIX_STEP_01_ONSP : BOOL;
   MIX_FWD_SS : BOOL;
   MIX_CYC_TIME_ACC : DINT;
   MIX_CYC_TIME : REAL;
   MIX_FWD_DEG : REAL;
   MIX_DEG_PER_SEC : REAL;
   MIX_STEP_02_ION : BOOL;   // REVERSE
   FWD_CMD_BON : TIMER := (PRE := 10000, ACC := 10002);
   REV_CMD_BON : TIMER := (PRE := 10000);
   LEFT_RIGHT_ENCODER_ERROR_DEG_REAL : REAL; {access None}
END_VAR

ROUTINE Logic   (* ladder *)
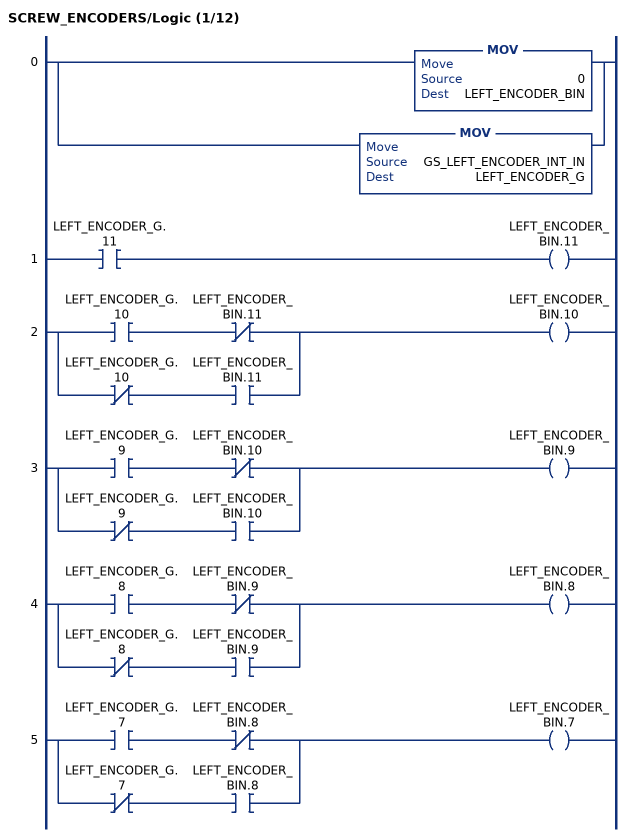
   0: [MOV(0,LEFT_ENCODER_BIN) ,MOV(GS_LEFT_ENCODER_INT_IN,LEFT_ENCODER_G) ];
   1: XIC(LEFT_ENCODER_G.11)OTE(LEFT_ENCODER_BIN.11);
   2: [XIC(LEFT_ENCODER_G.10) XIO(LEFT_ENCODER_BIN.11) ,XIO(LEFT_ENCODER_G.10) XIC(LEFT_ENCODER_BIN.11) ]OTE(LEFT_ENCODER_BIN.10);
   3: [XIC(LEFT_ENCODER_G.9) XIO(LEFT_ENCODER_BIN.10) ,XIO(LEFT_ENCODER_G.9) XIC(LEFT_ENCODER_BIN.10) ]OTE(LEFT_ENCODER_BIN.9);
   4: [XIC(LEFT_ENCODER_G.8) XIO(LEFT_ENCODER_BIN.9) ,XIO(LEFT_ENCODER_G.8) XIC(LEFT_ENCODER_BIN.9) ]OTE(LEFT_ENCODER_BIN.8);
   5: [XIC(LEFT_ENCODER_G.7) XIO(LEFT_ENCODER_BIN.8) ,XIO(LEFT_ENCODER_G.7) XIC(LEFT_ENCODER_BIN.8) ]OTE(LEFT_ENCODER_BIN.7);
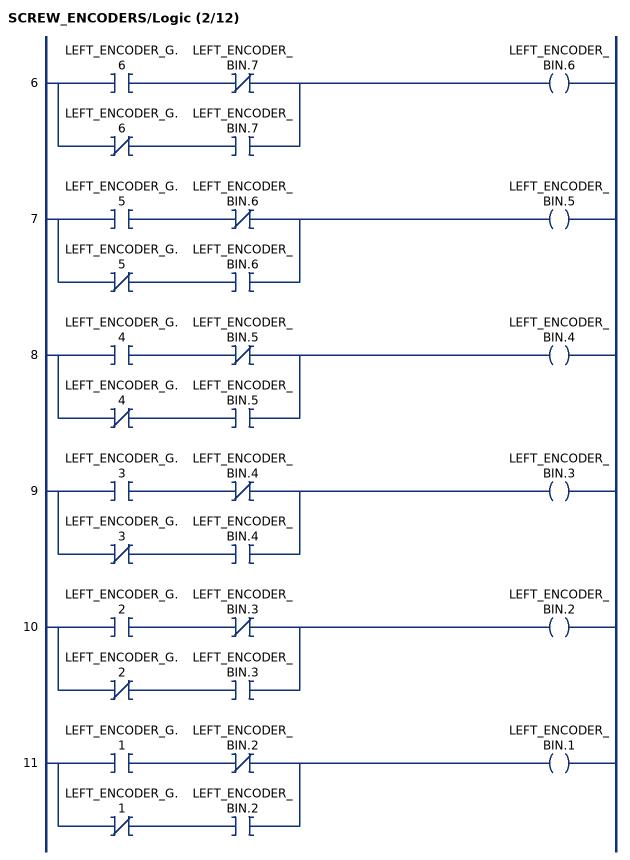
   6: [XIC(LEFT_ENCODER_G.6) XIO(LEFT_ENCODER_BIN.7) ,XIO(LEFT_ENCODER_G.6) XIC(LEFT_ENCODER_BIN.7) ]OTE(LEFT_ENCODER_BIN.6);
   7: [XIC(LEFT_ENCODER_G.5) XIO(LEFT_ENCODER_BIN.6) ,XIO(LEFT_ENCODER_G.5) XIC(LEFT_ENCODER_BIN.6) ]OTE(LEFT_ENCODER_BIN.5);
   8: [XIC(LEFT_ENCODER_G.4) XIO(LEFT_ENCODER_BIN.5) ,XIO(LEFT_ENCODER_G.4) XIC(LEFT_ENCODER_BIN.5) ]OTE(LEFT_ENCODER_BIN.4);
   9: [XIC(LEFT_ENCODER_G.3) XIO(LEFT_ENCODER_BIN.4) ,XIO(LEFT_ENCODER_G.3) XIC(LEFT_ENCODER_BIN.4) ]OTE(LEFT_ENCODER_BIN.3);
   10: [XIC(LEFT_ENCODER_G.2) XIO(LEFT_ENCODER_BIN.3) ,XIO(LEFT_ENCODER_G.2) XIC(LEFT_ENCODER_BIN.3) ]OTE(LEFT_ENCODER_BIN.2);
   11: [XIC(LEFT_ENCODER_G.1) XIO(LEFT_ENCODER_BIN.2) ,XIO(LEFT_ENCODER_G.1) XIC(LEFT_ENCODER_BIN.2) ]OTE(LEFT_ENCODER_BIN.1);
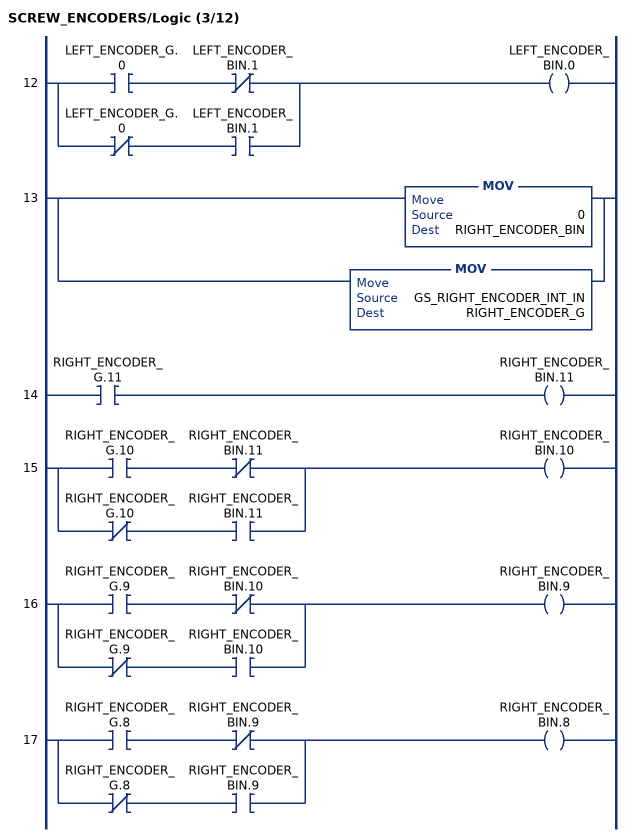
   12: [XIC(LEFT_ENCODER_G.0) XIO(LEFT_ENCODER_BIN.1) ,XIO(LEFT_ENCODER_G.0) XIC(LEFT_ENCODER_BIN.1) ]OTE(LEFT_ENCODER_BIN.0);
   13: [MOV(0,RIGHT_ENCODER_BIN) ,MOV(GS_RIGHT_ENCODER_INT_IN,RIGHT_ENCODER_G) ];
   14: XIC(RIGHT_ENCODER_G.11)OTE(RIGHT_ENCODER_BIN.11);
   15: [XIC(RIGHT_ENCODER_G.10) XIO(RIGHT_ENCODER_BIN.11) ,XIO(RIGHT_ENCODER_G.10) XIC(RIGHT_ENCODER_BIN.11) ]OTE(RIGHT_ENCODER_BIN.10);
   16: [XIC(RIGHT_ENCODER_G.9) XIO(RIGHT_ENCODER_BIN.10) ,XIO(RIGHT_ENCODER_G.9) XIC(RIGHT_ENCODER_BIN.10) ]OTE(RIGHT_ENCODER_BIN.9);
   17: [XIC(RIGHT_ENCODER_G.8) XIO(RIGHT_ENCODER_BIN.9) ,XIO(RIGHT_ENCODER_G.8) XIC(RIGHT_ENCODER_BIN.9) ]OTE(RIGHT_ENCODER_BIN.8);
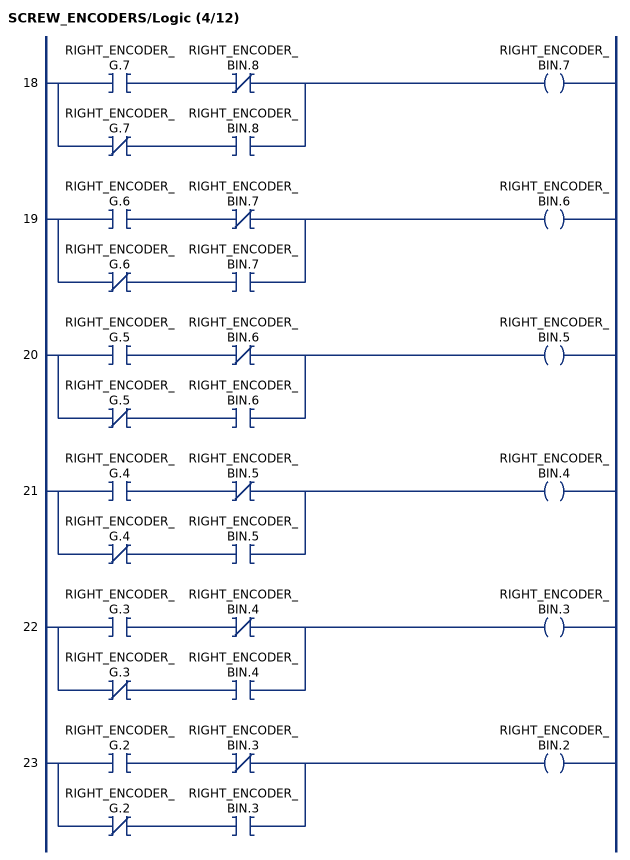
   18: [XIC(RIGHT_ENCODER_G.7) XIO(RIGHT_ENCODER_BIN.8) ,XIO(RIGHT_ENCODER_G.7) XIC(RIGHT_ENCODER_BIN.8) ]OTE(RIGHT_ENCODER_BIN.7);
   19: [XIC(RIGHT_ENCODER_G.6) XIO(RIGHT_ENCODER_BIN.7) ,XIO(RIGHT_ENCODER_G.6) XIC(RIGHT_ENCODER_BIN.7) ]OTE(RIGHT_ENCODER_BIN.6);
   20: [XIC(RIGHT_ENCODER_G.5) XIO(RIGHT_ENCODER_BIN.6) ,XIO(RIGHT_ENCODER_G.5) XIC(RIGHT_ENCODER_BIN.6) ]OTE(RIGHT_ENCODER_BIN.5);
   21: [XIC(RIGHT_ENCODER_G.4) XIO(RIGHT_ENCODER_BIN.5) ,XIO(RIGHT_ENCODER_G.4) XIC(RIGHT_ENCODER_BIN.5) ]OTE(RIGHT_ENCODER_BIN.4);
   22: [XIC(RIGHT_ENCODER_G.3) XIO(RIGHT_ENCODER_BIN.4) ,XIO(RIGHT_ENCODER_G.3) XIC(RIGHT_ENCODER_BIN.4) ]OTE(RIGHT_ENCODER_BIN.3);
   23: [XIC(RIGHT_ENCODER_G.2) XIO(RIGHT_ENCODER_BIN.3) ,XIO(RIGHT_ENCODER_G.2) XIC(RIGHT_ENCODER_BIN.3) ]OTE(RIGHT_ENCODER_BIN.2);
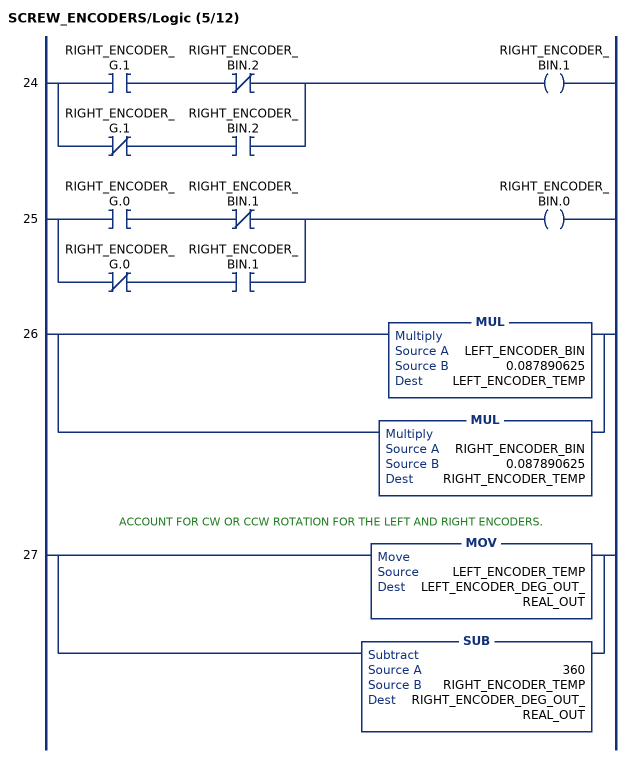
   24: [XIC(RIGHT_ENCODER_G.1) XIO(RIGHT_ENCODER_BIN.2) ,XIO(RIGHT_ENCODER_G.1) XIC(RIGHT_ENCODER_BIN.2) ]OTE(RIGHT_ENCODER_BIN.1);
   25: [XIC(RIGHT_ENCODER_G.0) XIO(RIGHT_ENCODER_BIN.1) ,XIO(RIGHT_ENCODER_G.0) XIC(RIGHT_ENCODER_BIN.1) ]OTE(RIGHT_ENCODER_BIN.0);
   26: [MUL(LEFT_ENCODER_BIN,0.087890625,LEFT_ENCODER_TEMP) ,MUL(RIGHT_ENCODER_BIN,0.087890625,RIGHT_ENCODER_TEMP) ];
   // ACCOUNT FOR CW OR CCW ROTATION FOR THE LEFT AND RIGHT ENCODERS.
   27: [MOV(LEFT_ENCODER_TEMP,LEFT_ENCODER_DEG_OUT_REAL_OUT) ,SUB(360,RIGHT_ENCODER_TEMP,RIGHT_ENCODER_DEG_OUT_REAL_OUT) ];
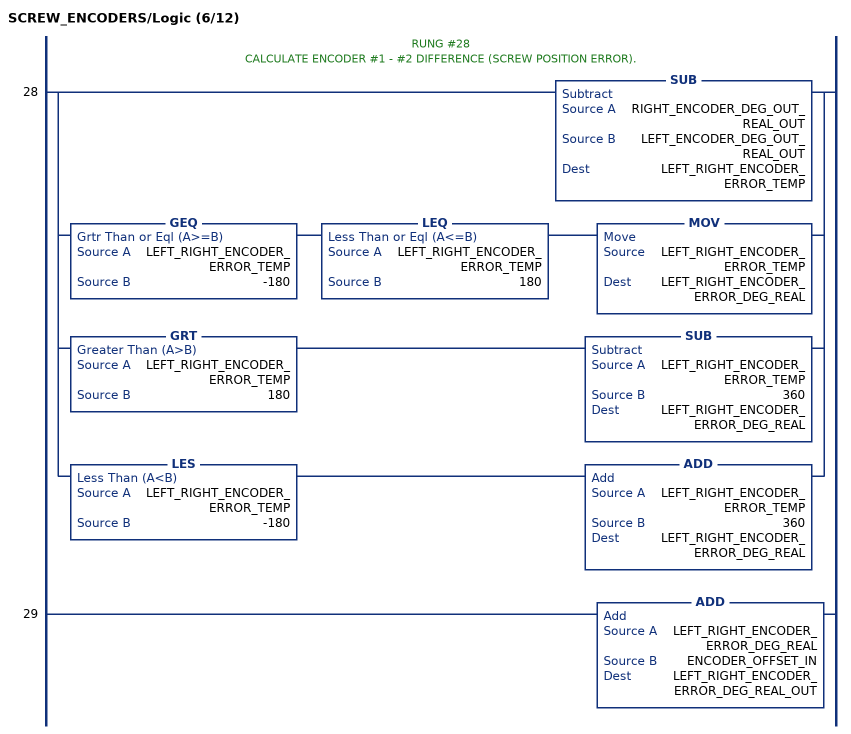
   // RUNG #28
   // CALCULATE ENCODER #1 - #2 DIFFERENCE (SCREW POSITION ERROR).
   28: [SUB(RIGHT_ENCODER_DEG_OUT_REAL_OUT,LEFT_ENCODER_DEG_OUT_REAL_OUT,LEFT_RIGHT_ENCODER_ERROR_TEMP) ,GEQ(LEFT_RIGHT_ENCODER_ERROR_TEMP,-180) LEQ(LEFT_RIGHT_ENCODER_ERROR_TEMP,180) MOV(LEFT_RIGHT_ENCODER_ERROR_TEMP,LEFT_RIGHT_ENCODER_ERROR_DEG_REAL) ,GRT(LEFT_RIGHT_ENCODER_ERROR_TEMP,180) SUB(LEFT_RIGHT_ENCODER_ERROR_TEMP,360,LEFT_RIGHT_ENCODER_ERROR_DEG_REAL) ,LES(LEFT_RIGHT_ENCODER_ERROR_TEMP,-180) ADD(LEFT_RIGHT_ENCODER_ERROR_TEMP,360,LEFT_RIGHT_ENCODER_ERROR_DEG_REAL) ];
   29: ADD(LEFT_RIGHT_ENCODER_ERROR_DEG_REAL,ENCODER_OFFSET_IN,LEFT_RIGHT_ENCODER_ERROR_DEG_REAL_OUT);
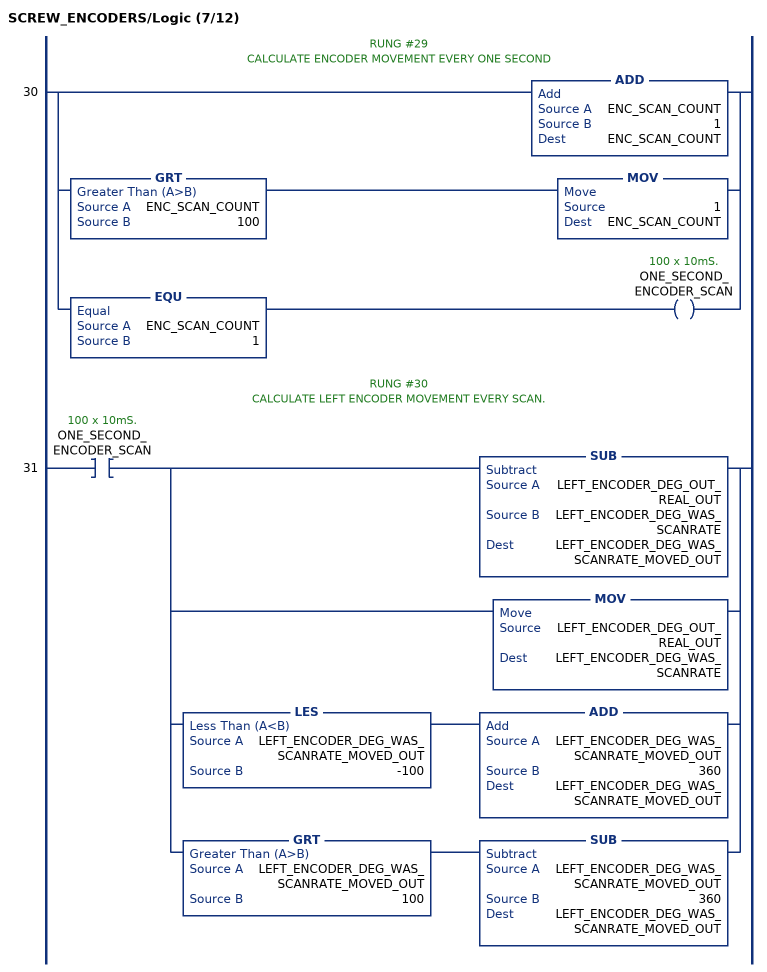
   // RUNG #29
   // CALCULATE ENCODER MOVEMENT EVERY ONE SECOND
   30: [ADD(ENC_SCAN_COUNT,1,ENC_SCAN_COUNT) ,GRT(ENC_SCAN_COUNT,100) MOV(1,ENC_SCAN_COUNT) ,EQU(ENC_SCAN_COUNT,1) OTE(ONE_SECOND_ENCODER_SCAN) ];
   // RUNG #30
   // CALCULATE LEFT ENCODER MOVEMENT EVERY SCAN.
   31: XIC(ONE_SECOND_ENCODER_SCAN)[SUB(LEFT_ENCODER_DEG_OUT_REAL_OUT,LEFT_ENCODER_DEG_WAS_SCANRATE,LEFT_ENCODER_DEG_WAS_SCANRATE_MOVED_OUT) ,MOV(LEFT_ENCODER_DEG_OUT_REAL_OUT,LEFT_ENCODER_DEG_WAS_SCANRATE) ,LES(LEFT_ENCODER_DEG_WAS_SCANRATE_MOVED_OUT,-100) ADD(LEFT_ENCODER_DEG_WAS_SCANRATE_MOVED_OUT,360,LEFT_ENCODER_DEG_WAS_SCANRATE_MOVED_OUT) ,GRT(LEFT_ENCODER_DEG_WAS_SCANRATE_MOVED_OUT,100) SUB(LEFT_ENCODER_DEG_WAS_SCANRATE_MOVED_OUT,360,LEFT_ENCODER_DEG_WAS_SCANRATE_MOVED_OUT) ];
